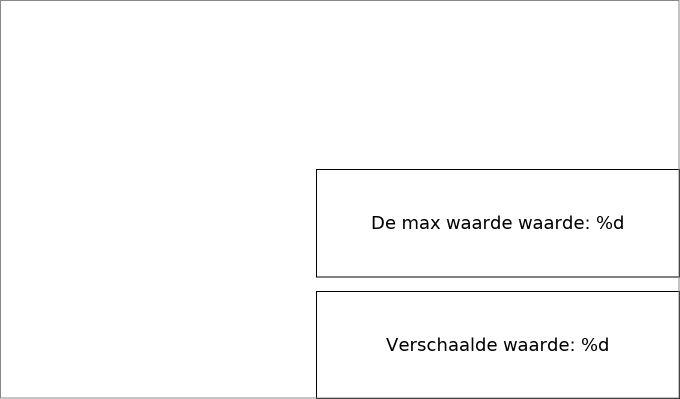
VISUALIZATION Visualization_DynamischVerschalen  // 680x399
    Rectangle (316,291 364x108), "Verschaalde waarde: %d", text variable: prg_DynamischVerschalen.nWaarde
    Rectangle (316,169 364x108), "De max waarde waarde: %d", text variable: prg_DynamischVerschalen.nScaledMax
        OnMouseDown: write the text variable via Default
END_VISUALIZATION

(* stored: Version 1.1.0.1, ProductVersion 3.1.4024.15
   Visu Visualization_DynamischVerschalen: Id {7924b989-dd9a-4b84-8916-200848775596} *)
